{library PUBLIC}
TYPE ABB_STATUS_OPERATING_MODE :
(
	ABB_STATUS_OPERATION_UNDEF:=0,				(* Undefined operating mode *)
	ABB_STATUS_OPERATION_AUTO:=1,				(* Automatic operating mode *)
	ABB_STATUS_OPERATION_MAN_PROG:=2, 			(* Manual operating mode MAX. 250 mm/S *)
	ABB_STATUS_OPERATION_MAN_TEST:=3 			(* Manual operating mode full speed, 100 % *)
);
END_TYPE

(* stored: Version 1.1.0.1, ProductVersion 3.1.4024.2
   EnumerationTextList ABB_STATUS_OPERATING_MODE: Id {31515297-df46-4726-bb3f-1d5e3a29d256} *)
